# EPICS substitutions: IOCs/12id/iocBoot/ioc12idd/picMot.substitutions
file "$(IP)/ipApp/Db/picos.db"
{
pattern
{P,      pChan,       DESC,          serChan }
{12idd:, 	 111,         pMotor111,        1    }
{12idd:, 	 112,         pMotor112,        1    }
{12idd:, 	 113,         pMotor113,        1    }

{12idd:, 	 121,         pMotor121,        1    }
{12idd:, 	 122,         pMotor122,        1    }
{12idd:, 	 123,         pMotor123,        1    }

{12idd:, 	 131,         pMotor131,        1    }
{12idd:, 	 132,         pMotor132,        1    }
{12idd:, 	 133,         pMotor133,        1    }

{12idd:, 	 141,         pMotor141,        1    }
{12idd:, 	 142,         pMotor142,        1    }
{12idd:, 	 143,         pMotor143,        1    }

{12idd:, 	 211,         pMotor211,        1    }
{12idd:, 	 212,         pMotor212,        1    }
{12idd:, 	 213,         pMotor213,        1    }

{12idd:, 	 221,         pMotor221,        1    }
{12idd:, 	 222,         pMotor222,        1    }
{12idd:, 	 223,         pMotor223,        1    }

{12idd:, 	 231,         pMotor231,        1    }
{12idd:, 	 232,         pMotor232,        1    }
{12idd:, 	 233,         pMotor233,        1    }

{12idd:, 	 241,         pMotor241,        1    }
{12idd:, 	 242,         pMotor242,        1    }
{12idd:, 	 243,         pMotor243,        1    }

}
